Fanuc KAREL source: kc00029.KL

-- PROVISIONAL review KL for V1013-1; original PC SHA256 94839238129d3a416759245b747002a4ed42c27fdff1df7cf35975671e3cae74
-- Incomplete behavior may be omitted. Consult companion uncertainty JSON. Do not deploy.
PROGRAM KC00029
%NOLOCKGROUP
BEGIN
  -- UNRESOLVED_PC offsets 5-17; opcodes 3F,75
  -- UNRESOLVED_PC offsets 22-106; opcodes 27,22,2A,22,22,22,22,22,22,22,22,22,22,22,22,31
  -- UNRESOLVED_PC offsets 111-115; opcodes 7F
END KC00029
